FUNCTION Convert_TOD_TO_STRING : Hresult
VAR_INPUT
	in : TOD;
	out : REFERENCE TO STRING;
END_VAR
VAR
	converted : STRING;
END_VAR
VAR CONSTANT
	INCOMPATIBLE : HRESULT := 16#9811070E;
END_VAR

converted := TOD_TO_STRING(in);

IF (STRING_TO_TOD(converted) <> in) THEN
	Convert_TOD_TO_STRING := INCOMPATIBLE;
	RETURN;
END_IF

out := converted;

END_FUNCTION

(* stored: Version 1.1.0.1, ProductVersion 3.1.4024.12
   POU Convert_TOD_TO_STRING: Id {d04c64ba-c5f6-44c3-a1de-f0af94d5cae4}, SpecialFunc None *)
